FUNCTION_BLOCK SL_MoveNeedleDown (* MoveNeedleDown: Requires NOT (AtTop AND AtBottom); Ensures (Position >= Distance) OR AtBottom; Invariant NOT (AtTop AND AtBottom); holds NeedleAxis.Down while running *)
  (* Standard: 61499-2 *)
  (* Version 0.1, 2026-09-28, Project contributors, AAU Smart Production Lab *)
  PACKAGE filler;
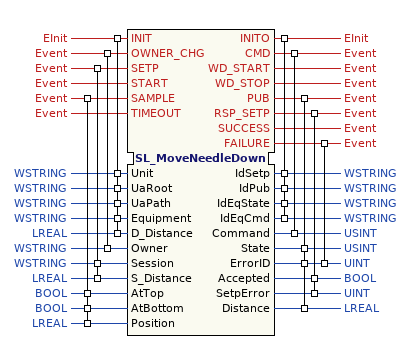
  EVENT_INPUT
    INIT : EInit WITH Unit, UaRoot, UaPath, Equipment, D_Distance;
    OWNER_CHG WITH Owner;
    SETP WITH Session, S_Distance;
    START;
    SAMPLE WITH AtTop, AtBottom, Position;
    TIMEOUT;
  END_EVENT
  EVENT_OUTPUT
    INITO : EInit WITH IdSetp, IdPub, IdEqState, IdEqCmd;
    CMD WITH Command;
    WD_START;
    WD_STOP;
    PUB WITH State, ErrorID, Distance;
    RSP_SETP WITH Accepted, SetpError;
    SUCCESS;
    FAILURE WITH ErrorID;
  END_EVENT
  VAR_INPUT
    Unit : WSTRING;
    UaRoot : WSTRING;
    UaPath : WSTRING;
    Equipment : WSTRING;
    D_Distance : LREAL;
    Owner : WSTRING;
    Session : WSTRING;
    S_Distance : LREAL;
    AtTop : BOOL;
    AtBottom : BOOL;
    Position : LREAL;
  END_VAR
  VAR_OUTPUT
    IdSetp : WSTRING;
    IdPub : WSTRING;
    IdEqState : WSTRING;
    IdEqCmd : WSTRING;
    Command : USINT;
    State : USINT;
    ErrorID : UINT;
    Accepted : BOOL;
    SetpError : UINT;
    Distance : LREAL := 50.0;
  END_VAR
  VAR
    Owned : BOOL;
    InRange : BOOL;
  END_VAR
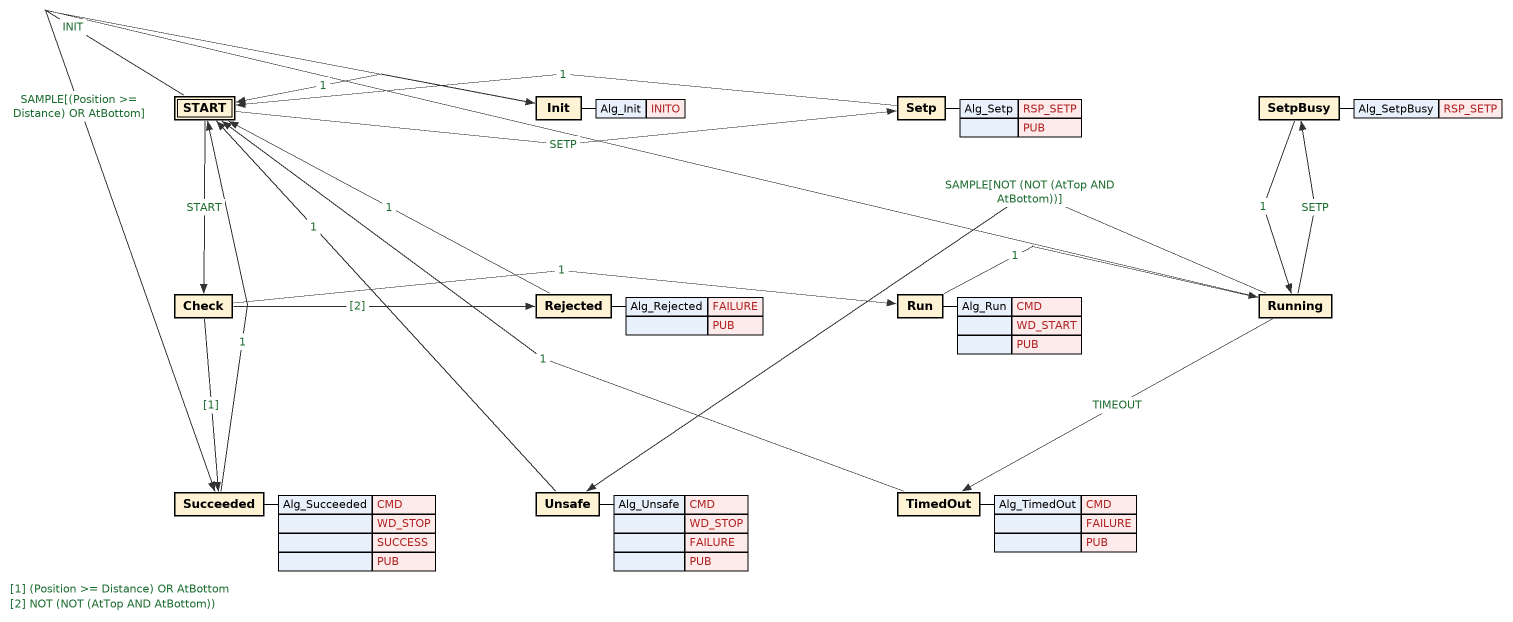
  EC_STATES
    START;
    Init : Alg_Init -> INITO;
    Setp : Alg_Setp -> RSP_SETP, -> PUB;
    SetpBusy : Alg_SetpBusy -> RSP_SETP;
    Check;
    Rejected : Alg_Rejected -> FAILURE, -> PUB;
    Run : Alg_Run -> CMD, -> WD_START, -> PUB;
    Running;
    Succeeded : Alg_Succeeded -> CMD, -> WD_STOP, -> SUCCESS, -> PUB;
    Unsafe : Alg_Unsafe -> CMD, -> WD_STOP, -> FAILURE, -> PUB;
    TimedOut : Alg_TimedOut -> CMD, -> FAILURE, -> PUB;
  END_STATES
  EC_TRANSITIONS
    START TO Init := INIT;
    START TO Setp := SETP;
    START TO Check := START;
    Check TO Rejected := NOT (NOT (AtTop AND AtBottom));
    Check TO Succeeded := (Position >= Distance) OR AtBottom;
    Check TO Run := 1;
    Run TO Running := 1;
    Running TO Unsafe := SAMPLE[NOT (NOT (AtTop AND AtBottom))];
    Running TO Succeeded := SAMPLE[(Position >= Distance) OR AtBottom];
    Running TO TimedOut := TIMEOUT;
    Running TO SetpBusy := SETP;
    SetpBusy TO Running := 1;
    Init TO START := 1;
    Setp TO START := 1;
    Rejected TO START := 1;
    Succeeded TO START := 1;
    Unsafe TO START := 1;
    TimedOut TO START := 1;
  END_TRANSITIONS
  ALGORITHM Alg_Init IN ST:
IdSetp := CONCAT(CONCAT("opc_ua[CREATE_METHOD;", CONCAT(UaRoot, UaPath)), "/SetParameters]");
IdPub := CONCAT(CONCAT(CONCAT(CONCAT(CONCAT(CONCAT(CONCAT(CONCAT("opc_ua[WRITE;", CONCAT(UaRoot, UaPath)), "/State;"), CONCAT(UaRoot, UaPath)), "/ErrorID"), ";"), CONCAT(UaRoot, UaPath)), "/Parameters/Distance"), "]");
IdEqState := CONCAT(CONCAT(CONCAT(CONCAT("loc[", Unit), "/"), Equipment), "/state]");
IdEqCmd := CONCAT(CONCAT(CONCAT(CONCAT("loc[", Unit), "/"), Equipment), "/cmd]");
Distance := D_Distance;
State := 0;
ErrorID := 0;
  END_ALGORITHM
  ALGORITHM Alg_Setp IN ST:
Owned := (Session = Owner) AND (Owner <> "");
InRange := (S_Distance >= 0.0) AND (S_Distance <= 50.0);
Accepted := FALSE;
IF NOT Owned THEN
  SetpError := 5;
ELSIF NOT InRange THEN
  SetpError := 8;
ELSE
  Distance := S_Distance;
  Accepted := TRUE;
  SetpError := 0;
END_IF;
  END_ALGORITHM
  ALGORITHM Alg_SetpBusy IN ST:
Accepted := FALSE;
SetpError := 6;
  END_ALGORITHM
  ALGORITHM Alg_Rejected IN ST:
State := 3;
ErrorID := 1;
  END_ALGORITHM
  ALGORITHM Alg_Run IN ST:
Command := 1;
State := 1;
ErrorID := 0;
  END_ALGORITHM
  ALGORITHM Alg_Succeeded IN ST:
Command := 0;
State := 2;
ErrorID := 0;
  END_ALGORITHM
  ALGORITHM Alg_Unsafe IN ST:
Command := 0;
State := 3;
ErrorID := 2;
  END_ALGORITHM
  ALGORITHM Alg_TimedOut IN ST:
Command := 0;
State := 3;
ErrorID := 3;
  END_ALGORITHM
END_FUNCTION_BLOCK
